Universal Robots URScript: 00B_03_JieXian_BiRang.script

def P00B_03_JieXian_BiRang():
  set_standard_analog_input_domain(0, 1)
  set_standard_analog_input_domain(1, 1)
  set_tool_analog_input_domain(0, 1)
  set_tool_analog_input_domain(1, 1)
  set_analog_outputdomain(0, 0)
  set_analog_outputdomain(1, 0)
  set_tool_voltage(0)
  set_input_actions_to_default()
  set_tcp(p[-0.06448999999999999,0.0207,0.28314999999999996,0.0,0.0,1.5902])
  set_payload(8.0)
  set_safety_mode_transition_hardness(1)
  set_gravity([0.0, 0.0, 9.82])
  $ 1 "机器人程序"
  $ 2 "MoveJ"
  $ 3 "路点_1"
  set_tcp(p[-0.06448999999999999,0.0207,0.28314999999999996,0.0,0.0,1.5902])
  movej(get_inverse_kin(p[.837498135851, -.258855992339, .722302211801, -.104209757527, .076877477528, -1.683818551649], qnear=[-0.16116649309267217, -1.816584889088766, -1.8520024458514612, -1.153778378163473, -1.608046833668844, 2.589193820953369]), a=0.6981317007977318, v=0.5235987755982988)
  $ 4 "路点_2"
  set_tcp(p[-0.06448999999999999,0.0207,0.28314999999999996,0.0,0.0,1.5902])
  movej(get_inverse_kin(p[.959228493109, -.089887190089, -.342497708464, -.476080577861, .477647347913, -1.502512602446], qnear=[0.1298479586839676, -3.310723129902975, -1.4381731192218226, -0.5691388289081019, -1.5120123068438929, 1.4643797874450684]), a=0.6981317007977318, v=0.5235987755982988)
end
